{attribute 'qualified_only'}
{attribute 'strict'}
TYPE E_StateType :
(
	Idle,
	Filling,
	Washing,
	Draining,
	Rinse,
	Completed
);
END_TYPE

(* stored: Version 1.1.0.1, ProductVersion 3.1.4024.16
   DUT E_StateType: Id {8a4c545b-7e59-4d6b-8563-7ee4a42fcbd1} *)
